// TIA Portal project "Blinking indicator lights - Course Problem #2" (V17)
// Problem Statement
// Blinking indicator lights are used quite extensively in industry. Design a circuit in which light is flashed after every 2 seconds.

(* hardware
DEVICE "S7-1200 station_1"  S7-1200 Station
   slot 0: "Rack_0"  S7-1200 Rack  Rack  V1.0
   slot 1: "PLC_1"  CPU 1215C DC/DC/Rly  6ES7 215-1HG40-0XB0  V4.5
*)

// ===== PLC "PLC_1"  CPU 1215C DC/DC/Rly =====

VAR_GLOBAL   // PLC tag table "Default tag table"
   "Start PB" AT %I0.0 : Bool;
   "Reset PB" AT %I0.1 : Bool;
   "Light" AT %Q0.0 : Bool;
   "Tag_1" AT %M0.0 : Bool;
END_VAR

// folder: System blocks/Program resources

DATA_BLOCK "IEC_Timer_0_DB"   // DB1
{ S7_Optimized_Access := 'TRUE' }
AUTHOR : Simatic
FAMILY : IEC
NAME : IEC_TMR
VERSION : 1.0
// stored: InstanceOfName IEC_TIMER
"IEC_TIMER"
BEGIN
END_DATA_BLOCK

DATA_BLOCK "IEC_Timer_0_DB_1"   // DB2
{ S7_Optimized_Access := 'TRUE' }
AUTHOR : Simatic
FAMILY : IEC
NAME : IEC_TMR
VERSION : 1.0
// stored: InstanceOfName IEC_TIMER
"IEC_TIMER"
BEGIN
END_DATA_BLOCK

// folder: (top level)

ORGANIZATION_BLOCK "Main"   // OB1, LAD, ProgramCycle
TITLE = "Main Program Sweep (Cycle)"
{ S7_Optimized_Access := 'TRUE' }
VERSION : 0.1
   VAR_INPUT
      Initial_Call : Bool;   // Initial call of this OB
      Remanence : Bool;   // =True, if remanent data are available
   END_VAR
BEGIN

REGION Network 1
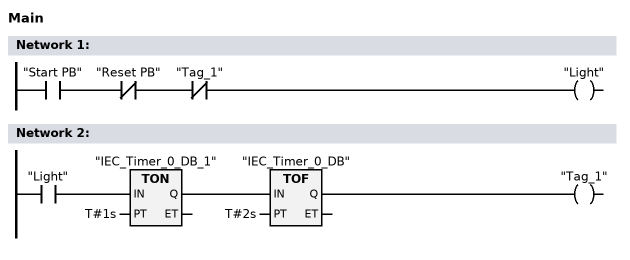
   RUNG wire#powerrail
      Contact( "Start PB" )
      I_Contact( "Reset PB" )
      I_Contact( "Tag_1" )
      Coil( "Light" )
   END_RUNG
   // the same network as SCL:
   "Light" := "Start PB" AND NOT "Reset PB" AND NOT "Tag_1";
END_REGION

REGION Network 2
   "IEC_Timer_0_DB_1".TON(IN := "Light", PT := T#1s);
   "IEC_Timer_0_DB".TOF(IN := "IEC_Timer_0_DB_1".Q, PT := T#2s);
   "Tag_1" := "IEC_Timer_0_DB".Q;
END_REGION
END_ORGANIZATION_BLOCK